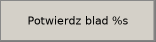
VISUALIZATION PIM_Confirm  // 156x42
VAR_IN_OUT
	fbStation:fbPIM_Station_V3;
END_VAR
    Button (0,0 156x42), "Potwierdz blad %s", text variable: fbStation.sStationName, invisible if: NOT fbStation.stPimInOut.bAlarmPLC AND NOT fbStation.stPimInOut.bWorkBlock_PLC AND fbStation.stPimInOut.sErrorCodePLC = ''
        OnMouseClick: execute {
            fbStation.stPimInOut.bNonBlockingAlarm := fbStation.stPimInOut.bAlarmPLC := fbStation.stPimInOut.bWorkBlock_PLC := FALSE;
            fbStation.stPimInOut.sErrorCodePLC := '';
            fbStation.stPimInOut.bConfirmEvent := TRUE;
        }
END_VISUALIZATION

(* stored: Version 1.1.0.1, ProductVersion 3.1.4024.12
   Visu PIM_Confirm: Id {6b199bb6-dd9a-4070-b76d-4558918acd2d} *)
